FUNCTION_BLOCK RFC_TransferWorkpieceTo_LSC EXTENDS RFC_MoveWorkpiece_Base
VAR_INPUT
END_VAR
VAR_OUTPUT
END_VAR
VAR
	// (EProcessVariables.LSC_ProductType = 0) AND ((EProcessVariables.RFC_WPAtEnd = TRUE) AND ((EProcessVariables.Crane_AtLSC = FALSE) OR ((EProcessVariables.Crane_AtLSC = TRUE) AND ((EProcessVariables.Crane_CylinderRetracted = TRUE) AND (EProcessVariables.Crane_HoldingWorkpiece = FALSE)))))
	m_compExpr203: ComparisonExpression(EProcessVariables.LSC_ProductType, EComparisonType.equals, EDataType.numeric, FALSE, 0, '', TRUE);
	m_compExpr205: ComparisonExpression(EProcessVariables.RFC_WPAtEnd, EComparisonType.equals, EDataType.binary, TRUE, 0, '', TRUE);
	m_compExpr207: ComparisonExpression(EProcessVariables.Crane_AtLSC, EComparisonType.equals, EDataType.binary, FALSE, 0, '', TRUE);
	m_compExpr209: ComparisonExpression(EProcessVariables.Crane_AtLSC, EComparisonType.equals, EDataType.binary, TRUE, 0, '', TRUE);
	m_compExpr211: ComparisonExpression(EProcessVariables.Crane_CylinderRetracted, EComparisonType.equals, EDataType.binary, TRUE, 0, '', TRUE);
	m_compExpr213: ComparisonExpression(EProcessVariables.Crane_HoldingWorkpiece, EComparisonType.equals, EDataType.binary, FALSE, 0, '', TRUE);
	m_boolExpr214: BoolExpression(m_compExpr211, EBoolOperation.and_op, m_compExpr213);
	m_boolExpr215: BoolExpression(m_compExpr209, EBoolOperation.and_op, m_boolExpr214);
	m_boolExpr216: BoolExpression(m_compExpr207, EBoolOperation.or_op, m_boolExpr215);
	m_boolExpr217: BoolExpression(m_compExpr205, EBoolOperation.and_op, m_boolExpr216);
	m_precondition: BoolExpression(m_compExpr203, EBoolOperation.and_op, m_boolExpr217);
	
	// EProcessVariables.RFC_SwitchRetracted = TRUE
	m_postcondition: ComparisonExpression(EProcessVariables.RFC_SwitchRetracted, EComparisonType.equals, EDataType.binary, TRUE, 0, '', TRUE);
		
	m_case: UINT := 0;
	m_timer: TON;
END_VAR

SUPER^();

METHOD PROTECTED  AtTarget : BOOL
VAR_INPUT
END_VAR
AtTarget := FALSE;

CASE m_case OF
	0:
		m_ptrRFC^.METH_Switch_Extend();
		m_timer(IN := TRUE, PT := T#200MS);
		IF m_timer.Q THEN
			m_case := 1;
			m_timer(IN := FALSE);
		END_IF
	
	1:
		m_ptrRFC^.METH_Switch_Retract();
		m_timer(IN := TRUE, PT := T#1000MS);
		IF m_timer.Q THEN
			m_case := 0;
			m_timer(IN := FALSE);
			AtTarget := TRUE;
		END_IF
	
END_CASE
END_METHOD

METHOD FB_init : BOOL
VAR_INPUT
	bInitRetains : BOOL; // if TRUE, the retain variables are initialized (warm start / cold start)
	bInCopyCode : BOOL;  // if TRUE, the instance afterwards gets moved into the copy code (online change)
	
	i_ptrRFC: POINTER TO RefeedingConveyor;
END_VAR
m_ptrRFC := i_ptrRFC;

m_id := EPrimitives.RFC_TransferWorkpieceTo_LSC;
m_timeout := T#200S;

Precondition := m_precondition;
Postcondition := m_postcondition;
END_METHOD

END_FUNCTION_BLOCK

(* stored: Version 1.1.0.1
   POU RFC_TransferWorkpieceTo_LSC: Id {493b710d-78d9-4a22-a962-84d030ce2fb5}, SpecialFunc None
   Method AtTarget: Id {1fc8613d-3613-47db-87b3-d935f3ab01dc}
   Method FB_init: Id {7e760f20-491f-41f6-a3b2-8c41e2a352d6} *)
